FUNCTION_BLOCK UDINT_AUDI_NE (* not equal *)
  (* Standard: 61131-3; Classification: standard comparison function; Description: Copyright (c) 2013 TU Wien ACIN\n \nThis program and the accompanying materials are made\navailable under the terms of the Eclipse Public License 2.0\nwhich is available at https://www.eclipse.org/legal/epl-2.0/\n\nSPDX-License-Identifier: EPL-2.0 *)
  (* Version 3.0, 2025-04-14, Patrick Aigner, changed package *)
  (* Version 1.0, 2013-03-13, Monika Wenger, TU Wien ACIN *)
  PACKAGE adapter::iec61131::comparison;
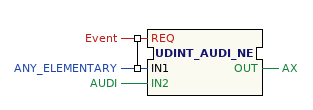
  EVENT_INPUT
    REQ WITH IN1; (* Service Request *)
  END_EVENT
  VAR_INPUT
    IN1 : ANY_ELEMENTARY; (* Input value 1 *)
  END_VAR
  SOCKETS
    IN2 : adapter::types::unidirectional::AUDI; (* Input value 2 *)
  END_SOCKETS
  PLUGS
    OUT : adapter::types::unidirectional::AX; (* value 1 != value2 = true *)
  END_PLUGS
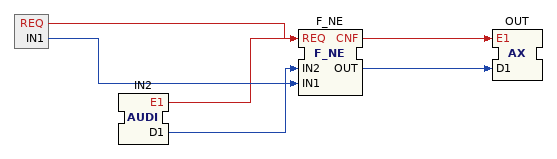
  FBS
    F_NE : iec61131::comparison::F_NE;
  END_FBS
  EVENT_CONNECTIONS
    F_NE.CNF TO OUT.E1;
    IN2.E1 TO F_NE.REQ;
    REQ TO F_NE.REQ;
  END_CONNECTIONS
  DATA_CONNECTIONS
    F_NE.OUT TO OUT.D1;
    IN2.D1 TO F_NE.IN2;
    IN1 TO F_NE.IN1;
  END_CONNECTIONS
END_FUNCTION_BLOCK
